ABB RobotStudio station: Pick_And_Place.rsstn

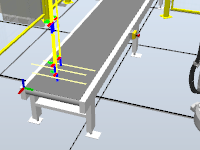
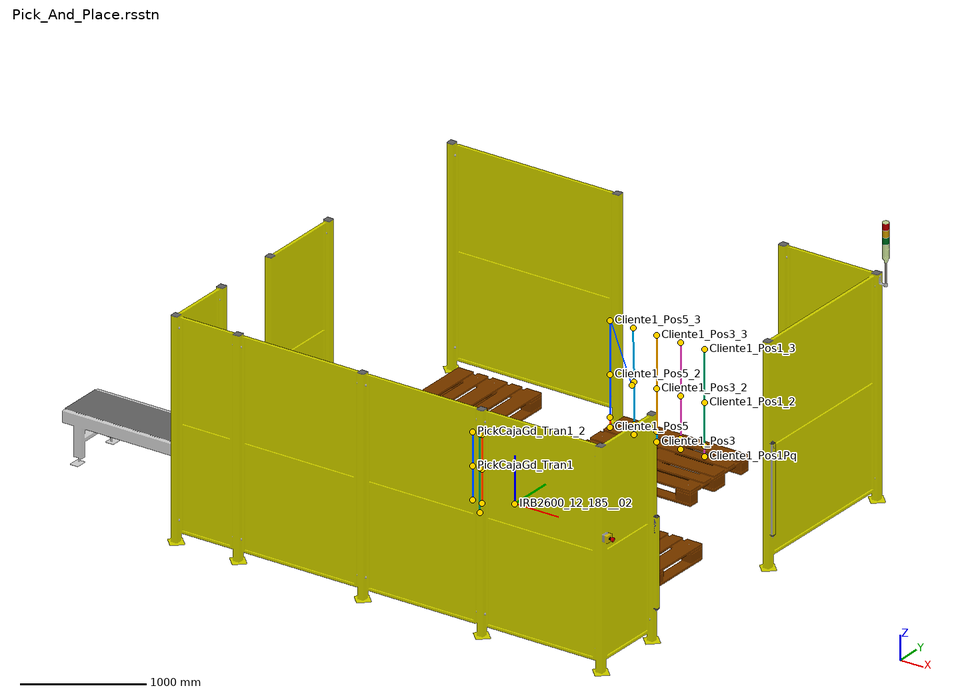
[picture v1: parts stored in the station drawn from their meshes, with robot base, taught points and paths (robot models come from the ABB library and are not in the file)]
Station Pick_1500V (saved by RobotStudio 22.1.9826.0)
Controller IRB2600_12_185
  mechanical unit ROB_1: IRB2600_12_185__02, 6 joints, base frame (0, 0, 0) mm
Layout (positions relative to the parent item):
  - IRB2600_12_185__02 [mechanism, from Robots\IRB2600_12_185_G_02.rslib] at (0, 0, 0) mm; joint values [0, 0, 0, 0, 0.5236, 0] (rad or m)
  - euro pallet [part] at (580, 1100, 0) mm, rotated rx 0 ry 0 rz 90 deg, size 803.9 x 1205.8 x 151.5 mm
  - euro pallet_2 [part] at (1400, -600, 0) mm, size 803.9 x 1205.8 x 151.5 mm
  - euro pallet_3 [part] at (-1200, 900, 0) mm, size 803.9 x 1205.8 x 151.5 mm
  - SC_VentosaTool [smart component] at (1018.61, 0, 1417.5) mm, rotated rx 180 ry 60 rz 180 deg
      signals: DI DI_Attacher
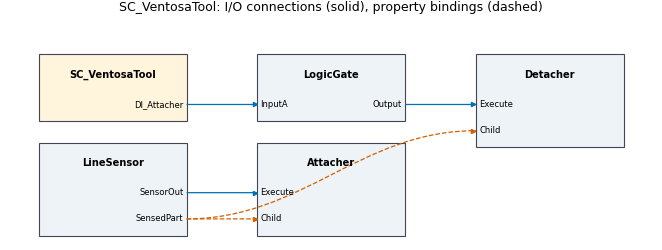
      connections:
        SC_VentosaTool.DI_Attacher -> LogicGate.InputA
        LogicGate.Output -> Detacher.Execute
        LineSensor.SensorOut -> Attacher.Execute
        LineSensor.SensedPart => Attacher.Child
        LineSensor.SensedPart => Detacher.Child
    - Ventosa_Tool [mechanism, from Libraries\Ventosa_Tool.rslib] at (0, 0, 0) mm
    - Attacher [smart component, from Components\Attacher.rslib]
        properties: Parent=Ventosa_Tool; Flange=0; Child=(none); Mount=false; Offset=[0 0 0]; Orientation=[0 0 0]
    - Detacher [smart component, from Components\Detacher.rslib]
        properties: Child=(none); KeepPosition=true
    - LineSensor [smart component, from Components\LineSensor.rslib]
        properties: Start=[0 0 0.1255]; End=[0 0 0.1555]; Radius=0.001; SensedPart=(none); SensedPoint=[0 0 0]
      - _sensorPart_ [part], size 2 x 2 x 30 mm
    - LogicGate [smart component, from Components\LogicGate.rslib]
        properties: Operator=NOT; Delay=0
  - 950_4000_h2_2 [part, from Equipment\Conveyor 950 4000 h2.rslib] at (-3500, -1800, 0) mm
  - SC_Conveyor [smart component]
      signals: DI Crear_Caja_Pq, DI Crear_CajaGd, DO DO_Sensor, DI Crear_Caja_Md, DO DO_Sensor2, DO DO_Sensor3
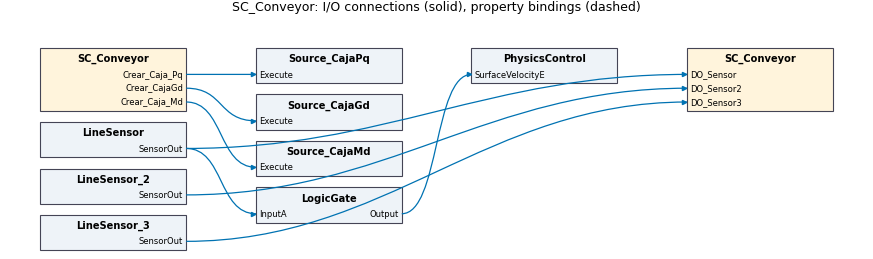
      connections:
        SC_Conveyor.Crear_Caja_Pq -> Source_CajaPq.Execute
        SC_Conveyor.Crear_CajaGd -> Source_CajaGd.Execute
        SC_Conveyor.Crear_Caja_Md -> Source_CajaMd.Execute
        LineSensor.SensorOut -> SC_Conveyor.DO_Sensor
        LineSensor.SensorOut -> LogicGate.InputA
        LogicGate.Output -> PhysicsControl.SurfaceVelocityEnabled
        LineSensor_2.SensorOut -> SC_Conveyor.DO_Sensor2
        LineSensor_3.SensorOut -> SC_Conveyor.DO_Sensor3
    - Cinta [part] at (-3400, -1350, 425) mm, size 4000 x 415.7 x 2 mm
    - CajaPq [part] at (-3400, -1243.92, 515.9) mm, size 203.3 x 177.8 x 88.9 mm
    - CajaMd [part] at (-3400, -1243.92, 604.8) mm, size 203.2 x 177.8 x 177.8 mm
    - CajaGd [part] at (-3400, -1243.92, 604.8) mm, size 355.6 x 177.8 x 177.8 mm
    - Source_CajaPq [smart component, from Components\Source.rslib]
        properties: Source=CajaPq; Copy=(none); Parent=(none); Position=[-3.4 -1.24392 0.5159]; Orientation=[0 0 0]; Transient=true; PhysicsBehavior=3
    - Source_CajaMd [smart component, from Components\Source.rslib]
        properties: Source=CajaMd; Copy=(none); Parent=(none); Position=[-3.4 -1.24392 0.6048]; Orientation=[0 0 0]; Transient=true; PhysicsBehavior=3
    - Source_CajaGd [smart component, from Components\Source.rslib]
        properties: Source=CajaGd; Copy=(none); Parent=(none); Position=[-3.4 -1.24392 0.6048]; Orientation=[0 0 0]; Transient=true; PhysicsBehavior=3
    - PhysicsControl [smart component, from Components\PhysicsControl.rslib]
        properties: Object=Cinta; Behavior=1; SurfaceVelocity=1
    - LineSensor [smart component, from Components\LineSensor.rslib]
        properties: Start=[0.475 -0.93427 0.475]; End=[0.475 -1.35 0.475]; Radius=0; SensedPart=(none); SensedPoint=[0 0 0]
      - _sensorPart_ [part], size 0 x 415.7 x 0 mm
    - LogicGate [smart component, from Components\LogicGate.rslib]
        properties: Operator=NOT; Delay=0
    - LineSensor_2 [smart component, from Components\LineSensor.rslib]
        properties: Start=[0.475 -0.93427 0.55]; End=[0.475 -1.35 0.55]; Radius=0; SensedPart=(none); SensedPoint=[0 0 0]
      - _sensorPart_ [part], size 0 x 415.7 x 0 mm
    - LineSensor_3 [smart component, from Components\LineSensor.rslib]
        properties: Start=[0.3 -0.93427 0.475]; End=[0.3 -1.35 0.475]; Radius=0; SensedPart=(none); SensedPoint=[0 0 0]
      - _sensorPart_ [part], size 0 x 415.7 x 0 mm
  - IRC5_Control-Module [part, from Equipment\IRC5_Control-Module.rslib] at (-1550, -2600, 0) mm, rotated rx 90 ry 0 rz 0 deg
  - Fence [graphiccomponentgroup]
    - Segment 1 [part], size 169.7 x 169.7 x 2000 mm
    - Segment 2 [part], size 1234.9 x 169.7 x 2000 mm
    - Segment 2 [part], size 1234.9 x 169.7 x 2000 mm
    - Segment 3 [part], size 1284.9 x 169.7 x 2000 mm
  - Fence [graphiccomponentgroup]
    - Segment 1 [part], size 169.7 x 169.7 x 2000 mm
    - Segment 2 [part], size 169.7 x 784.9 x 2000 mm
  - Fence [graphiccomponentgroup]
    - Segment 1 [part], size 169.7 x 169.7 x 2000 mm
    - Segment 2 [part], size 169.7 x 1584.9 x 2000 mm
    - Segment 3 [part], size 984.9 x 169.7 x 2000 mm
  - Fence [graphiccomponentgroup]
    - Segment 1 [part], size 169.7 x 169.7 x 2000 mm
    - Segment 2 [part], size 1684.9 x 169.7 x 2000 mm
  - Fence [graphiccomponentgroup]
    - Segment 1 [part], size 169.7 x 169.7 x 2000 mm
    - Segment 2 [part], size 169.7 x 884.9 x 2000 mm
  - Fence [graphiccomponentgroup]
    - Segment 3 [part], size 684.9 x 169.7 x 2000 mm
  - Fence [graphiccomponentgroup]
    - Segment 3 [part], size 684.9 x 169.7 x 2000 mm
  - Roller Conveyor [part], size 4000 x 588 x 420 mm
  - Fence [graphiccomponentgroup]
    - Segment 1 [part], size 169.7 x 169.7 x 2000 mm
    - Segment 2 [part], size 169.7 x 714.3 x 2000 mm
  - Fence [graphiccomponentgroup]
    - Segment 1 [part], size 169.7 x 169.7 x 2000 mm
    - Segment 2 [part], size 169.7 x 714.3 x 2000 mm
  - Baliza [part] at (2062, 1410, 1800) mm, rotated rx 90 ry 0 rz 90 deg, size 55 x 568.4 x 80.6 mm
  - Estop [part] at (2331, -2100, 1200) mm, rotated rx 0 ry 0 rz -90 deg, size 67 x 89.5 x 67 mm
  - Estop_2 [part] at (-1800, 1730, 1200) mm, size 67 x 89.5 x 67 mm
  - Estop_3 [part] at (-500, -900, 382) mm, size 67 x 89.5 x 67 mm
  - Cortina [part] at (2357, -1430, 300) mm, rotated rx 0 ry -90 rz 0 deg, size 845 x 30 x 36 mm
  - Cortina_2 [part] at (2362, 200, 300) mm, rotated rx 0 ry -90 rz 90 deg, size 845 x 30 x 36 mm
  - Sistema de coordenadas_2 [frame] at (0, 0, 125.5) mm
Attachment: SC_VentosaTool is attached to IRB2600_12_185__02 / Link6
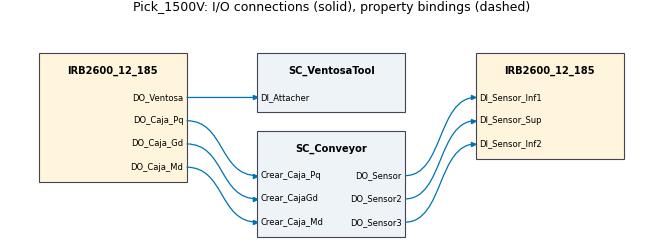
Station logic (signal -> signal, property => property):
  SC_Conveyor.DO_Sensor -> IRB2600_12_185.DI_Sensor_Inf1
  IRB2600_12_185.DO_Ventosa -> SC_VentosaTool.DI_Attacher
  IRB2600_12_185.DO_Caja_Pq -> SC_Conveyor.Crear_Caja_Pq
  IRB2600_12_185.DO_Caja_Gd -> SC_Conveyor.Crear_CajaGd
  IRB2600_12_185.DO_Caja_Md -> SC_Conveyor.Crear_Caja_Md
  SC_Conveyor.DO_Sensor2 -> IRB2600_12_185.DI_Sensor_Sup
  SC_Conveyor.DO_Sensor3 -> IRB2600_12_185.DI_Sensor_Inf2
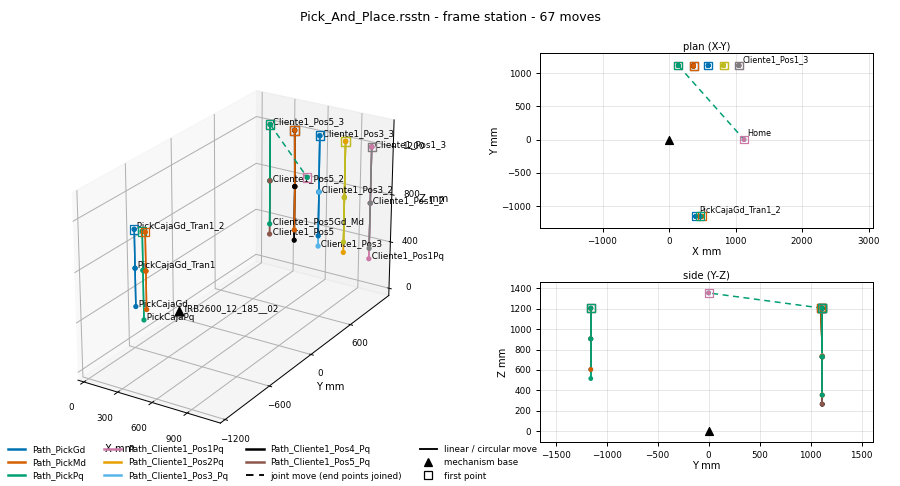
[picture p0: tool path of Pick_And_Place.rsstn in frame station, 67 of 67 moves have a stored position in this frame; points joined in program order, loops and branches not executed]
Targets, tools, work objects and paths stored in the station, written as RAPID:
! task T_ROB1
MODULE CalibData
  TASK PERS wobjdata WO_Pick:=[FALSE,TRUE,"",[[600,-1350,427],[1,0,0,0]],[[0,0,0],[1,0,0,0]]];
  TASK PERS wobjdata WO_Cliente:=[FALSE,TRUE,"",[[1200,700,23],[0.707107,0,0,0.707107]],[[0,0,0],[1,0,0,0]]];
  TASK PERS wobjdata WO_Cliente2:=[FALSE,TRUE,"",[[816,887,23],[1,0,0,0]],[[0,0,0],[1,0,0,0]]];
  TASK PERS wobjdata WO_Cliente3:=[FALSE,TRUE,"",[[411,1316,21],[1,0,0,0]],[[0,0,0],[1,0,0,0]]];
ENDMODULE

! task T_ROB1
MODULE Module1
  PERS tooldata TCP_Ventosa_Tool:=[TRUE,[[0,0,125.5],[1,0,0,0]],[0.93,[0.267,-0.58,58],[1,0,0,0],0,0,0]];
  CONST robtarget Home:=[[1127.298347497,0,1354.75],[0.5,0,0.866025404,0],[0,0,0,0],[9E+09,9E+09,9E+09,9E+09,9E+09,9E+09]];
  CONST robtarget PickCajaGd:=[[-198.25,194.98,177.8],[0,1,0,0],[-1,0,1,0],[9E+09,9E+09,9E+09,9E+09,9E+09,9E+09]];
  CONST robtarget PickCajaGd_Tran1:=[[-198.25,194.98,477.8],[0,1,0,0],[-1,0,1,0],[9E+09,9E+09,9E+09,9E+09,9E+09,9E+09]];
  CONST robtarget PickCajaGd_Tran1_2:=[[-198.25,194.98,777.8],[0,1,0,0],[0,0,0,0],[9E+09,9E+09,9E+09,9E+09,9E+09,9E+09]];
  CONST robtarget PickCajaMd:=[[-105.45,194.98,177.8],[0,1,0,0],[-1,0,1,0],[9E+09,9E+09,9E+09,9E+09,9E+09,9E+09]];
  CONST robtarget PickCajaMd_Tran1:=[[-105.45,194.98,477.8],[0,1,0,0],[-1,0,1,0],[9E+09,9E+09,9E+09,9E+09,9E+09,9E+09]];
  CONST robtarget PickCajaMd_Tran1_2:=[[-105.45,194.98,777.8],[0,1,0,0],[0,0,0,0],[9E+09,9E+09,9E+09,9E+09,9E+09,9E+09]];
  CONST robtarget PickCajaPq:=[[-130.35,194.98,88.9],[0,1,0,0],[0,0,0,0],[9E+09,9E+09,9E+09,9E+09,9E+09,9E+09]];
  CONST robtarget PickCajaPq_Tran1:=[[-130.45,194.98,477.8],[0,1,0,0],[-1,0,1,0],[9E+09,9E+09,9E+09,9E+09,9E+09,9E+09]];
  CONST robtarget PickCajaPq_Tran1_2:=[[-130.45,194.98,777.8],[0,1,0,0],[0,0,0,0],[9E+09,9E+09,9E+09,9E+09,9E+09,9E+09]];
  CONST robtarget Cliente1_Pos1Pq:=[[412.75,149.9,242],[0,1,0,0],[-1,0,1,0],[9E+09,9E+09,9E+09,9E+09,9E+09,9E+09]];
  CONST robtarget Cliente1_Pos1_2:=[[412.75,149.9,714.888633463],[0,1,0,0],[0,0,0,0],[9E+09,9E+09,9E+09,9E+09,9E+09,9E+09]];
  CONST robtarget Cliente1_Pos1_3:=[[412.75,149.9,1182.272966271],[0,1,0,0],[0,0,0,0],[9E+09,9E+09,9E+09,9E+09,9E+09,9E+09]];
  CONST robtarget Cliente1_Pos2:=[[412.75,379.9,242],[0,1,0,0],[-1,0,1,0],[9E+09,9E+09,9E+09,9E+09,9E+09,9E+09]];
  CONST robtarget Cliente1_Pos2_2:=[[412.75,379.9,711.545706382],[0,1,0,0],[-1,0,1,0],[9E+09,9E+09,9E+09,9E+09,9E+09,9E+09]];
  CONST robtarget Cliente1_Pos2_3:=[[412.75,379.9,1180.505219025],[0,1,0,0],[0,0,0,0],[9E+09,9E+09,9E+09,9E+09,9E+09,9E+09]];
  CONST robtarget Cliente1_Pos3:=[[412.75,609.9,242],[0,1,0,0],[-1,0,1,0],[9E+09,9E+09,9E+09,9E+09,9E+09,9E+09]];
  CONST robtarget Cliente1_Pos3_2:=[[412.75,609.9,707.203396556],[0,1,0,0],[0,0,0,0],[9E+09,9E+09,9E+09,9E+09,9E+09,9E+09]];
  CONST robtarget Cliente1_Pos3_3:=[[412.75,609.9,1179.988097675],[0,1,0,0],[0,0,0,0],[9E+09,9E+09,9E+09,9E+09,9E+09,9E+09]];
  CONST robtarget Cliente1_Pos4:=[[412.75,829.9,242],[0,1,0,0],[0,0,1,0],[9E+09,9E+09,9E+09,9E+09,9E+09,9E+09]];
  CONST robtarget Cliente1_Pos4_2:=[[412.75,829.9,705.416260416],[0,1,0,0],[0,0,1,0],[9E+09,9E+09,9E+09,9E+09,9E+09,9E+09]];
  CONST robtarget Cliente1_Pos4_3:=[[401.196074105,829.9,1183.950208913],[0,1,0,0],[0,0,1,0],[9E+09,9E+09,9E+09,9E+09,9E+09,9E+09]];
  CONST robtarget Cliente1_Pos5:=[[412.75,1059.9,242],[0,1,0,0],[0,0,1,0],[9E+09,9E+09,9E+09,9E+09,9E+09,9E+09]];
  CONST robtarget Cliente1_Pos5_2:=[[412.75,1059.9,704.273658884],[0,1,0,0],[0,0,1,0],[9E+09,9E+09,9E+09,9E+09,9E+09,9E+09]];
  CONST robtarget Cliente1_Pos5_3:=[[412.75,1059.9,1182.545603822],[0,1,0,0],[0,0,1,0],[9E+09,9E+09,9E+09,9E+09,9E+09,9E+09]];
  CONST robtarget Cliente1_Pos1Gd_Md:=[[412.75,149.9,330.9],[0,1,0,0],[-1,0,1,0],[9E+09,9E+09,9E+09,9E+09,9E+09,9E+09]];
  CONST robtarget Cliente1_Pos2Gd_Md:=[[412.75,379.9,330.9],[0,1,0,0],[-1,0,1,0],[9E+09,9E+09,9E+09,9E+09,9E+09,9E+09]];
  CONST robtarget Cliente1_Pos3Gd_Md:=[[412.75,609.9,330.9],[0,1,0,0],[-1,0,1,0],[9E+09,9E+09,9E+09,9E+09,9E+09,9E+09]];
  CONST robtarget Cliente1_Pos4Gd_Md:=[[412.75,829.9,330.9],[0,1,0,0],[0,0,1,0],[9E+09,9E+09,9E+09,9E+09,9E+09,9E+09]];
  CONST robtarget Cliente1_Pos5Gd_Md:=[[412.75,1059.9,330.9],[0,1,0,0],[0,0,1,0],[9E+09,9E+09,9E+09,9E+09,9E+09,9E+09]];
  PROC Path_PickGd()
    MoveJ PickCajaGd_Tran1_2,v1500,z100,TCP_Ventosa_Tool\WObj:=WO_Pick;
    MoveL PickCajaGd_Tran1,v1500,fine,TCP_Ventosa_Tool\WObj:=WO_Pick;
    MoveLDO PickCajaGd,v800,fine,TCP_Ventosa_Tool\WObj:=WO_Pick,DO_Ventosa,1;
    WaitTime 0.8;
    MoveL PickCajaGd_Tran1,v1500,fine,TCP_Ventosa_Tool\WObj:=WO_Pick;
    MoveL PickCajaGd_Tran1_2,v1500,z100,TCP_Ventosa_Tool\WObj:=WO_Pick;
  ENDPROC
  PROC Path_PickMd()
    MoveJ PickCajaMd_Tran1_2,v1500,z100,TCP_Ventosa_Tool\WObj:=WO_Pick;
    MoveL PickCajaMd_Tran1,v1500,z0,TCP_Ventosa_Tool\WObj:=WO_Pick;
    MoveLDO PickCajaMd,v800,z0,TCP_Ventosa_Tool\WObj:=WO_Pick,DO_Ventosa,1;
    WaitTime 0.8;
    MoveL PickCajaMd_Tran1,v1500,z0,TCP_Ventosa_Tool\WObj:=WO_Pick;
    MoveL PickCajaMd_Tran1_2,v1500,z100,TCP_Ventosa_Tool\WObj:=WO_Pick;
  ENDPROC
  PROC Path_PickPq()
    MoveJ PickCajaPq_Tran1_2,v1500,z100,TCP_Ventosa_Tool\WObj:=WO_Pick;
    MoveL PickCajaPq_Tran1,v1500,z0,TCP_Ventosa_Tool\WObj:=WO_Pick;
    MoveLDO PickCajaPq,v800,z0,TCP_Ventosa_Tool\WObj:=WO_Pick,DO_Ventosa,1;
    WaitTime 0.8;
    MoveL PickCajaPq_Tran1,v1500,z0,TCP_Ventosa_Tool\WObj:=WO_Pick;
    MoveL PickCajaPq_Tran1_2,v1500,z100,TCP_Ventosa_Tool\WObj:=WO_Pick;
  ENDPROC
  PROC Path_Cliente1_Pos1Pq()
    MoveJ Cliente1_Pos1_3,v1500,z100,TCP_Ventosa_Tool\WObj:=WO_Cliente;
    MoveL Cliente1_Pos1_2,v1500,z0,TCP_Ventosa_Tool\WObj:=WO_Cliente;
    MoveLDO Cliente1_Pos1Pq,v800,z0,TCP_Ventosa_Tool\WObj:=WO_Cliente,DO_Ventosa,0;
    WaitTime 0.8;
    MoveL Cliente1_Pos1_2,v1500,z0,TCP_Ventosa_Tool\WObj:=WO_Cliente;
    MoveL Cliente1_Pos1_3,v1500,z100,TCP_Ventosa_Tool\WObj:=WO_Cliente;
  ENDPROC
  PROC Path_Cliente1_Pos2Pq()
    MoveJ Cliente1_Pos2_3,v1500,z100,TCP_Ventosa_Tool\WObj:=WO_Cliente;
    MoveL Cliente1_Pos2_2,v1500,z0,TCP_Ventosa_Tool\WObj:=WO_Cliente;
    MoveLDO Cliente1_Pos2,v800,z0,TCP_Ventosa_Tool\WObj:=WO_Cliente,DO_Ventosa,0;
    WaitTime 0.8;
    MoveL Cliente1_Pos2_2,v1500,z0,TCP_Ventosa_Tool\WObj:=WO_Cliente;
    MoveL Cliente1_Pos2_3,v1500,z100,TCP_Ventosa_Tool\WObj:=WO_Cliente;
  ENDPROC
  PROC Path_Cliente1_Pos3_Pq()
    MoveJ Cliente1_Pos3_3,v1500,z100,TCP_Ventosa_Tool\WObj:=WO_Cliente;
    MoveL Cliente1_Pos3_2,v1500,z0,TCP_Ventosa_Tool\WObj:=WO_Cliente;
    MoveLDO Cliente1_Pos3,v800,z0,TCP_Ventosa_Tool\WObj:=WO_Cliente,DO_Ventosa,0;
    WaitTime 0.8;
    MoveL Cliente1_Pos3_2,v1500,z0,TCP_Ventosa_Tool\WObj:=WO_Cliente;
    MoveL Cliente1_Pos3_3,v1500,z100,TCP_Ventosa_Tool\WObj:=WO_Cliente;
  ENDPROC
  PROC Path_Cliente1_Pos4_Pq()
    MoveJ Cliente1_Pos4_3,v1500,z100,TCP_Ventosa_Tool\WObj:=WO_Cliente;
    MoveL Cliente1_Pos4_2,v1500,z0,TCP_Ventosa_Tool\WObj:=WO_Cliente;
    MoveLDO Cliente1_Pos4,v800,z0,TCP_Ventosa_Tool\WObj:=WO_Cliente,DO_Ventosa,0;
    WaitTime 0.8;
    MoveL Cliente1_Pos4_2,v1500,z0,TCP_Ventosa_Tool\WObj:=WO_Cliente;
    MoveL Cliente1_Pos4_3,v1500,z100,TCP_Ventosa_Tool\WObj:=WO_Cliente;
  ENDPROC
  PROC Path_Cliente1_Pos5_Pq()
    MoveJ Cliente1_Pos5_3,v1500,z100,TCP_Ventosa_Tool\WObj:=WO_Cliente;
    MoveL Cliente1_Pos5_2,v1500,z0,TCP_Ventosa_Tool\WObj:=WO_Cliente;
    MoveLDO Cliente1_Pos5,v800,z0,TCP_Ventosa_Tool\WObj:=WO_Cliente,DO_Ventosa,0;
    WaitTime 0.8;
    MoveL Cliente1_Pos5_2,v1500,z0,TCP_Ventosa_Tool\WObj:=WO_Cliente;
    MoveL Cliente1_Pos5_3,v1500,z100,TCP_Ventosa_Tool\WObj:=WO_Cliente;
  ENDPROC
  PROC Path_Cliente1_Pos1_GdMd()
    MoveJ Cliente1_Pos1_3,v1500,z100,TCP_Ventosa_Tool\WObj:=WO_Cliente;
    MoveL Cliente1_Pos1_2,v1500,z0,TCP_Ventosa_Tool\WObj:=WO_Cliente;
    MoveLDO Cliente1_Pos1Gd_Md,v800,z0,TCP_Ventosa_Tool\WObj:=WO_Cliente,DO_Ventosa,0;
    WaitTime 0.8;
    MoveL Cliente1_Pos1_2,v1500,z0,TCP_Ventosa_Tool\WObj:=WO_Cliente;
    MoveL Cliente1_Pos1_3,v1500,z100,TCP_Ventosa_Tool\WObj:=WO_Cliente;
  ENDPROC
  PROC Path_Cliente1_Pos2_GdMd()
    MoveJ Cliente1_Pos2_3,v1500,z100,TCP_Ventosa_Tool\WObj:=WO_Cliente;
    MoveL Cliente1_Pos2_2,v1500,z0,TCP_Ventosa_Tool\WObj:=WO_Cliente;
    MoveLDO Cliente1_Pos2Gd_Md,v800,z0,TCP_Ventosa_Tool\WObj:=WO_Cliente,DO_Ventosa,0;
    WaitTime 0.8;
    MoveL Cliente1_Pos2_2,v1500,z0,TCP_Ventosa_Tool\WObj:=WO_Cliente;
    MoveL Cliente1_Pos2_3,v1500,z100,TCP_Ventosa_Tool\WObj:=WO_Cliente;
  ENDPROC
  PROC Path_Cliente1_Pos3_GdMd()
    MoveJ Cliente1_Pos3_3,v1500,z100,TCP_Ventosa_Tool\WObj:=WO_Cliente;
    MoveL Cliente1_Pos3_2,v1500,z0,TCP_Ventosa_Tool\WObj:=WO_Cliente;
    MoveLDO Cliente1_Pos3Gd_Md,v800,z0,TCP_Ventosa_Tool\WObj:=WO_Cliente,DO_Ventosa,0;
    WaitTime 0.8;
    MoveL Cliente1_Pos3_2,v1500,z0,TCP_Ventosa_Tool\WObj:=WO_Cliente;
    MoveL Cliente1_Pos3_3,v1500,z100,TCP_Ventosa_Tool\WObj:=WO_Cliente;
  ENDPROC
  PROC Path_Cliente1_Pos4_GdMd()
    MoveJ Cliente1_Pos4_3,v1500,z100,TCP_Ventosa_Tool\WObj:=WO_Cliente;
    MoveL Cliente1_Pos4_2,v1500,z0,TCP_Ventosa_Tool\WObj:=WO_Cliente;
    MoveLDO Cliente1_Pos4Gd_Md,v800,z0,TCP_Ventosa_Tool\WObj:=WO_Cliente,DO_Ventosa,0;
    WaitTime 0.8;
    MoveL Cliente1_Pos4_2,v1500,z0,TCP_Ventosa_Tool\WObj:=WO_Cliente;
    MoveL Cliente1_Pos4_3,v1500,z100,TCP_Ventosa_Tool\WObj:=WO_Cliente;
  ENDPROC
  PROC Path_Cliente1_Pos5_GdMd()
    MoveJ Cliente1_Pos5_3,v1500,z100,TCP_Ventosa_Tool\WObj:=WO_Cliente;
    MoveL Cliente1_Pos5_2,v1500,z0,TCP_Ventosa_Tool\WObj:=WO_Cliente;
    MoveLDO Cliente1_Pos5Gd_Md,v800,z0,TCP_Ventosa_Tool\WObj:=WO_Cliente,DO_Ventosa,0;
    WaitTime 0.8;
    MoveL Cliente1_Pos5_2,v1500,z0,TCP_Ventosa_Tool\WObj:=WO_Cliente;
    MoveL Cliente1_Pos5_3,v1500,z100,TCP_Ventosa_Tool\WObj:=WO_Cliente;
    MoveJ Home,v800,z0,TCP_Ventosa_Tool\WObj:=wobj0;
  ENDPROC
  PROC main()
    MoveJ Home,v800,z0,TCP_Ventosa_Tool\WObj:=wobj0;
    Path_CajaPq;
    WaitTime 0.5;
    Path_CajaMd;
    WaitTime 0.5;
    Path_CajaGd;
    WaitTime 0.5;
  ENDPROC
  PROC Path_CajaGd()
    Path_PickGd;
    Path_Cliente1_Pos1_GdMd;
    Path_Cliente1_Pos2_GdMd;
    Path_Cliente1_Pos3_GdMd;
    Path_Cliente1_Pos4_GdMd;
    Path_Cliente1_Pos5_GdMd;
  ENDPROC
  PROC Path_CajaMd()
    Path_PickMd;
    Path_Cliente1_Pos1_GdMd;
    Path_Cliente1_Pos2_GdMd;
    Path_Cliente1_Pos3_GdMd;
    Path_Cliente1_Pos4_GdMd;
    Path_Cliente1_Pos5_GdMd;
  ENDPROC
  PROC Path_CajaPq()
    Path_PickPq;
    Path_Cliente1_Pos1Pq;
    Path_Cliente1_Pos2Pq;
    Path_Cliente1_Pos3_Pq;
    Path_Cliente1_Pos4_Pq;
    Path_Cliente1_Pos5_Pq;
  ENDPROC
ENDMODULE

